// Mitsubishi GX Works2 project: ProjectAtAll1 (1) (2)   PLC: FX3G

// global labels: Global1
VAR_GLOBAL
  Temperature_sensor AT X002 : BOOL;
  Flicking_light3 AT Y003 : BOOL;
  Working_light AT Y007 : BOOL;
  Empty_templets AT X003 : BOOL;
  Melting_Start AT X001 : BOOL;
  Melting_light AT Y001 : BOOL;
  Melting AT Y003 : BOOL;
END_VAR
VAR_GLOBAL CONSTANT
  Nuts_for_Nuts_Mix : REAL := 100;
  Pistachio_for_Nuts_Mix : REAL := 100;
  Nuts_for_Dubai_Chocolate : REAL := 20;
  Pistachio_for_Dubai_Chocolate : REAL := 120;
  Kadaif_for_Dubai_Chocolate : REAL := 60;
END_VAR
VAR_GLOBAL
  Choose_choclate_type AT X004 : BOOL;
END_VAR
VAR_GLOBAL CONSTANT
  Min_Input : INT;
END_VAR
VAR_GLOBAL
  Is_Nuts_Mix AT M150 : BOOL;
  Save_Analog AT D1180 : REAL;
  Analog_Input_1 AT D8280 : INT;
  Analog_Output_2 : BOOL;
  Nuts_Stock AT D1800 : REAL;
  Pistachio_Stock AT D1810 : REAL;
  Kadaif_Stock AT D1820 : REAL;
END_VAR
VAR_GLOBAL CONSTANT
  Melting_Container : REAL := 400;
END_VAR
VAR_GLOBAL
  New_Melting_Container AT D1200 : REAL;
  Empty_templete_sensor AT M3 : BOOL;
END_VAR
VAR_GLOBAL CONSTANT
  Trayes : INT := 4;
END_VAR
VAR_GLOBAL
  Mold_light AT Y002 : BOOL;
END_VAR
VAR_GLOBAL CONSTANT
  Times : INT := 40;
END_VAR
VAR_GLOBAL
  Pass_to_cold_system AT X006 : BOOL;
  Melting_Amount AT D1220 : REAL;
  Not_Enough_Stock AT M7 : BOOL;
  Start_day AT X007 : BOOL;
  Emergency_button AT X005 : BOOL;
  End_the_day AT M5 : BOOL;
  Initial_chocolate AT D1300 : REAL;
  Initial_nuts AT D1310 : REAL;
  Initial_pistachio AT D1320 : REAL;
  Initial_kadaif AT D1330 : REAL;
  Chocolate_Stock AT D1830 : REAL;
END_VAR
VAR_GLOBAL CONSTANT
  Min_Chocolat_Coins : REAL := 400;
END_VAR
VAR_GLOBAL
  Melting_Indicator AT M380 : BOOL;
  Mold_time AT TS4 : BOOL;
  Molding_four_seconds AT TC4 : BOOL;
END_VAR
VAR_GLOBAL CONSTANT
  Div_400_choclate_grams : REAL := 400;
END_VAR
VAR_GLOBAL
  Chocolate_Picked AT D1840 : REAL;
END_VAR
VAR_GLOBAL CONSTANT
  Dubai_Condition_At_Least_6 : REAL := 6;
  Nuts_Mix_Condition_Max_Val : REAL;
END_VAR
VAR_GLOBAL
  Dubai_Picked AT M6 : BOOL;
  Nuts_Mix_Picked AT M5 : BOOL;
END_VAR
VAR_GLOBAL CONSTANT
  Dubai_Condition_At_Least_5 : REAL := 5;
END_VAR
VAR_GLOBAL
  Dubai_chocolate_filling AT D1900 : REAL;
  Nuts_mix_chacolate_filling AT D1910 : REAL;
  Is_Working AT Y007 : BOOL;
  Filling_timer4 AT TC2 : BOOL;
  Filling_timer3 AT TC1 : BOOL;
END_VAR
VAR_GLOBAL CONSTANT
  Five_Second : INT := 50;
END_VAR
VAR_GLOBAL
  Filling_time AT TC1 : BOOL;
  Filling_time1 AT TS1 : BOOL;
  Filling_time2 AT TS2 : BOOL;
  Flicking_light4 AT Y004 : BOOL;
  Flickering_light_index AT M0 : BOOL;
  Count_five_seconds AT TC6 : BOOL;
END_VAR
VAR_GLOBAL CONSTANT
  half_of_Second : INT := 5;
END_VAR
VAR_GLOBAL
  Finish_five_seconds AT TS6 : BOOL;
  Dubai_choclate_frizzing AT D1500 : REAL;
  Nuts_mix_chocolate_frizzing AT D1510 : REAL;
  Freezing_three_seconds AT TC7 : BOOL;
END_VAR
VAR_GLOBAL CONSTANT
  Three_seconds_waiting : INT := 30;
END_VAR
VAR_GLOBAL
  Freezing_time AT TS7 : BOOL;
  Freezing_light AT Y006 : BOOL;
  Packeging_mechine AT D1600 : REAL;
  Dubai_packeging_mechine AT D1600 : REAL;
  Nuts_packeging_mechine AT D1610 : REAL;
END_VAR
VAR_GLOBAL CONSTANT
  Equals_four : REAL := 4;
END_VAR
VAR_GLOBAL
  Dubai_chocolata_bar AT D1700 : REAL;
  Nuts_chocolata_bar AT D1710 : REAL;
  Switch_choclate_table AT X000 : BOOL;
  End_package_light AT Y005 : BOOL;
  Dubai_package AT D1400 : REAL;
  Nuts_mix_package AT D1410 : REAL;
  Package_counter AT CC1 : BOOL;
END_VAR
VAR_GLOBAL CONSTANT
  Four_bars_for_package : INT := 4;
END_VAR
VAR_GLOBAL
  Package_indicator AT M10 : BOOL;
END_VAR
VAR_GLOBAL CONSTANT
  Zero : INT;
END_VAR
VAR_GLOBAL
  Package_indicator2 AT M11 : BOOL;
  Finish_freezing_indicator AT M8 : BOOL;
END_VAR
VAR_GLOBAL CONSTANT
  Three_bars_for_package : INT := 3;
END_VAR
VAR_GLOBAL
  Bars_in_package AT CN1 : INT;
  Package_ready AT CC1 : BOOL;
  Number_of_packages AT D1940 : REAL;
END_VAR
VAR_GLOBAL CONSTANT
  One_package : REAL := 1;
END_VAR
VAR_GLOBAL
  Finish_one_package AT M12 : BOOL;
  End_of_the_day_index AT M13 : BOOL;
END_VAR
VAR_GLOBAL CONSTANT
  Multipy_by_fourty : REAL := 40;
END_VAR
VAR_GLOBAL
  Number_of_packages_output AT D1950 : REAL;
  Analog_Output AT D8282 : INT;
END_VAR

// task Task_01 (event TRUE, interval 0, priority 31): POU_01

PROGRAM POU_01
VAR
  Analog_Output_1 : BOOL;
END_VAR
VAR CONSTANT
  Five_Seconds : INT := 50;
  half_Second : INT := 5;
END_VAR
(* structured ladder/FBD written out as ST: instructions are called as NAME(EN, inputs, outputs); _pN, _eN, _tN stand for wires *)
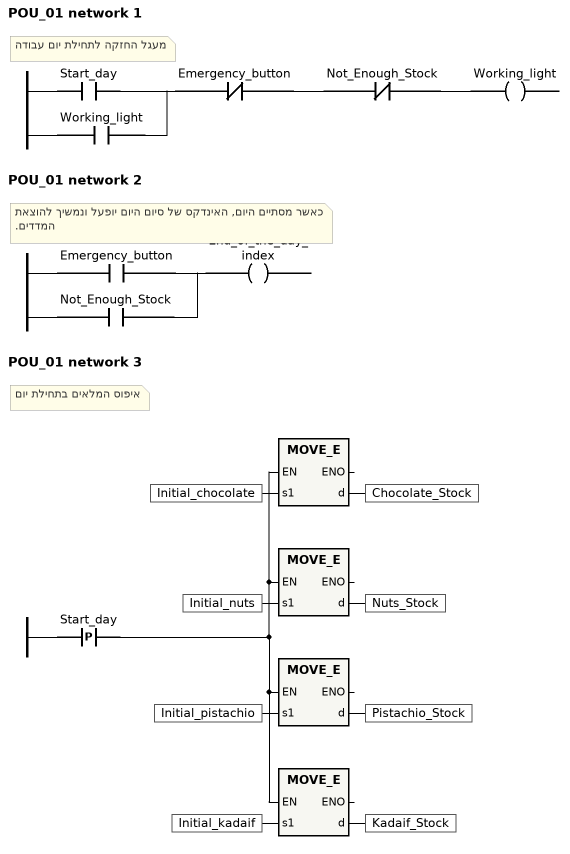
(* network 1 *)
(* מעגל החזקה לתחילת יום עבודה *)
Working_light := ((Start_day OR Working_light) AND NOT Emergency_button) AND NOT Not_Enough_Stock;
(* network 2 *)
(* כאשר מסתיים היום, האינדקס של סיום היום יופעל ונמשיך להוצאת המדדים. *)
End_of_the_day_index := Emergency_button OR Not_Enough_Stock;
(* network 3 *)
(* איפוס המלאים בתחילת יום *)
_p1 := LDP(TRUE, Start_day);
MOVE_E(_p1, Initial_chocolate, Chocolate_Stock);
MOVE_E(_p1, Initial_nuts, Nuts_Stock);
MOVE_E(_p1, Initial_pistachio, Pistachio_Stock);
MOVE_E(_p1, Initial_kadaif, Kadaif_Stock);
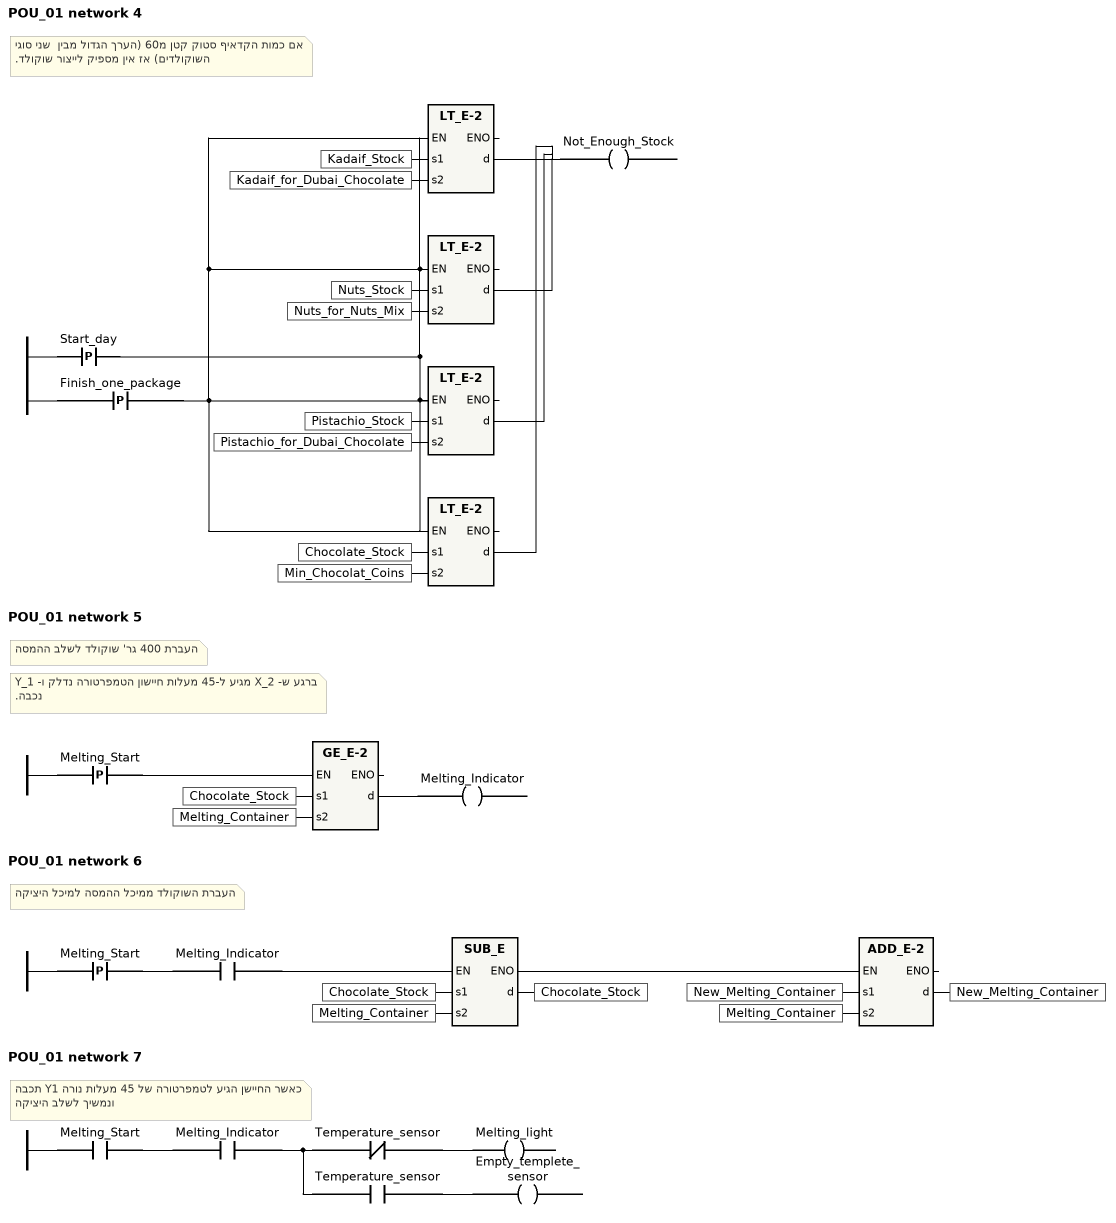
(* network 4 *)
(* אם כמות הקדאיף סטוק קטן מ60 (הערך הגדול מבין  שני סוגי השוקולדים) אז אין מספיק לייצור שוקולד. *)
_p1 := LDP(TRUE, Start_day) OR LDP(TRUE, Finish_one_package);
LT_E(_p1, Kadaif_Stock, Kadaif_for_Dubai_Chocolate, _t2);
LT_E(_p1, Nuts_Stock, Nuts_for_Nuts_Mix, _t3);
LT_E(_p1, Pistachio_Stock, Pistachio_for_Dubai_Chocolate, _t4);
LT_E(_p1, Chocolate_Stock, Min_Chocolat_Coins, _t5);
Not_Enough_Stock := _t2 OR _t3 OR _t4 OR _t5;
(* network 5 *)
(* העברת 400 גר' שוקולד לשלב ההמסה *)
(* ברגע ש- X_2 מגיע ל-45 מעלות חיישון הטמפרטורה נדלק ו- Y_1 נכבה. *)
GE_E(LDP(TRUE, Melting_Start), Chocolate_Stock, Melting_Container, _t1);
Melting_Indicator := _t1;
(* network 6 *)
(* העברת השוקולד ממיכל ההמסה למיכל היציקה *)
_e1 := SUB_E(LDP(TRUE, Melting_Start) AND Melting_Indicator, Chocolate_Stock, Melting_Container, Chocolate_Stock);
ADD_E(_e1, New_Melting_Container, Melting_Container, New_Melting_Container);
(* network 7 *)
(* כאשר החיישן הגיע לטמפרטורה של 45 מעלות נורה Y1 תכבה ונמשיך לשלב היציקה *)
_p1 := Melting_Start AND Melting_Indicator;
Melting_light := _p1 AND NOT Temperature_sensor;
Empty_templete_sensor := _p1 AND Temperature_sensor;
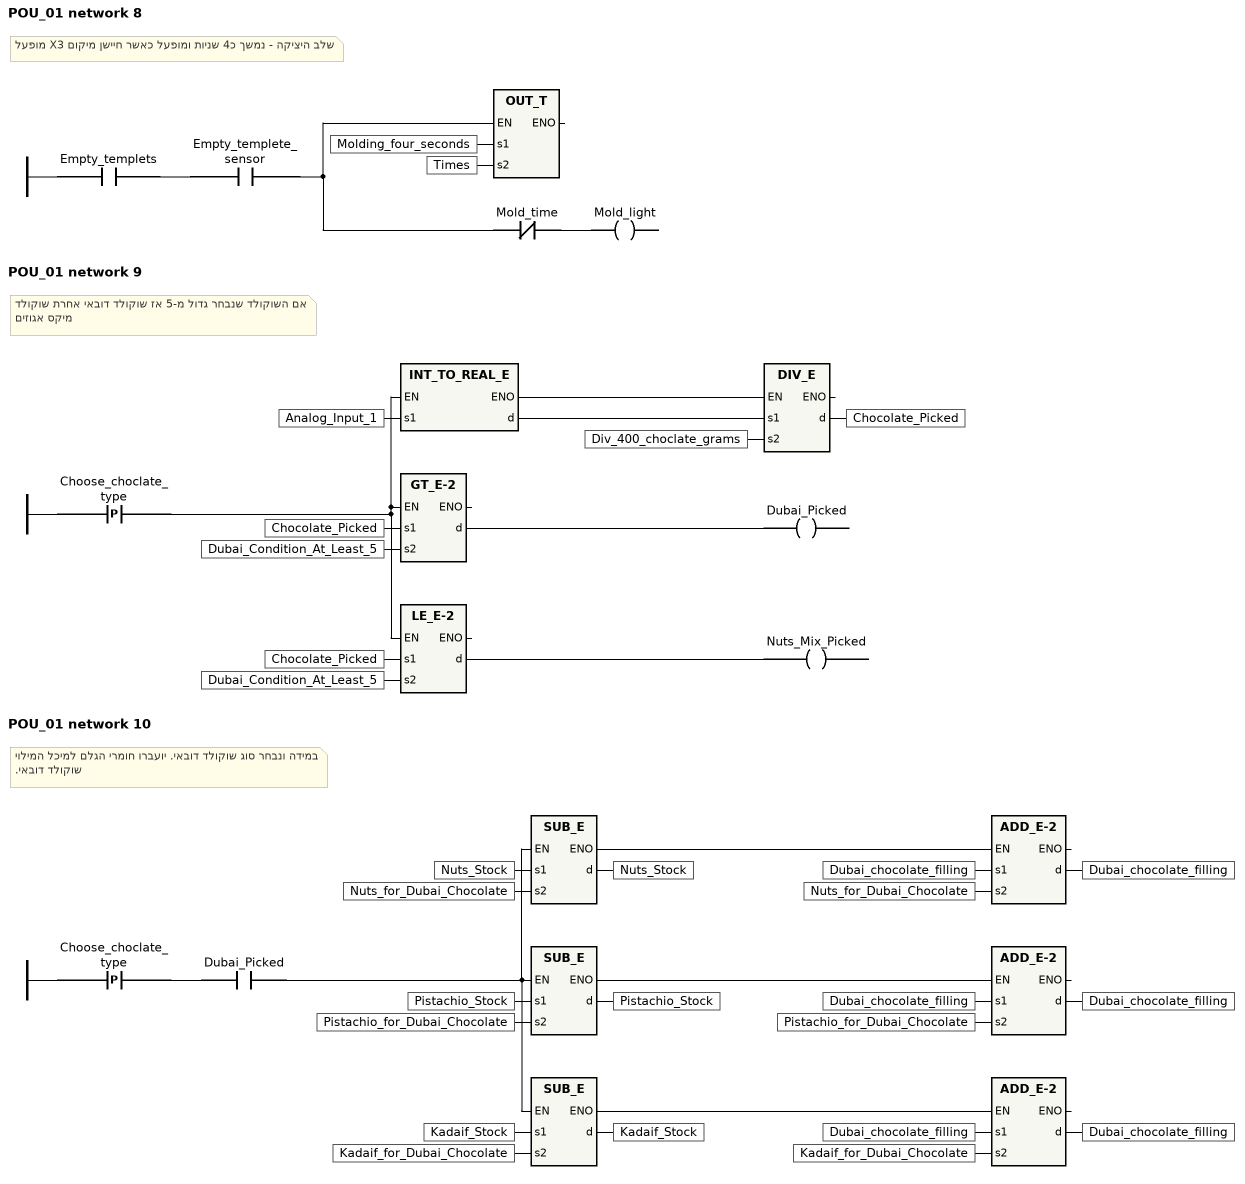
(* network 8 *)
(* שלב היציקה - נמשך כ4 שניות ומופעל כאשר חיישן מיקום X3 מופעל *)
_p1 := Empty_templets AND Empty_templete_sensor;
OUT_T(_p1, Molding_four_seconds, Times);
Mold_light := _p1 AND NOT Mold_time;
(* network 9 *)
(* אם השוקולד שנבחר גדול מ-5 אז שוקולד דובאי אחרת שוקולד מיקס אגוזים *)
_p1 := LDP(TRUE, Choose_choclate_type);
_e3 := INT_TO_REAL_E(_p1, Analog_Input_1, _t2);
DIV_E(_e3, _t2, Div_400_choclate_grams, Chocolate_Picked);
GT_E(_p1, Chocolate_Picked, Dubai_Condition_At_Least_5, _t4);
Dubai_Picked := _t4;
LE_E(_p1, Chocolate_Picked, Dubai_Condition_At_Least_5, _t5);
Nuts_Mix_Picked := _t5;
(* network 10 *)
(* במידה ונבחר סוג שוקולד דובאי. יועברו חומרי הגלם למיכל המילוי שוקולד דובאי. *)
_p1 := LDP(TRUE, Choose_choclate_type) AND Dubai_Picked;
_e2 := SUB_E(_p1, Nuts_Stock, Nuts_for_Dubai_Chocolate, Nuts_Stock);
ADD_E(_e2, Dubai_chocolate_filling, Nuts_for_Dubai_Chocolate, Dubai_chocolate_filling);
_e3 := SUB_E(_p1, Pistachio_Stock, Pistachio_for_Dubai_Chocolate, Pistachio_Stock);
ADD_E(_e3, Dubai_chocolate_filling, Pistachio_for_Dubai_Chocolate, Dubai_chocolate_filling);
_e4 := SUB_E(_p1, Kadaif_Stock, Kadaif_for_Dubai_Chocolate, Kadaif_Stock);
ADD_E(_e4, Dubai_chocolate_filling, Kadaif_for_Dubai_Chocolate, Dubai_chocolate_filling);
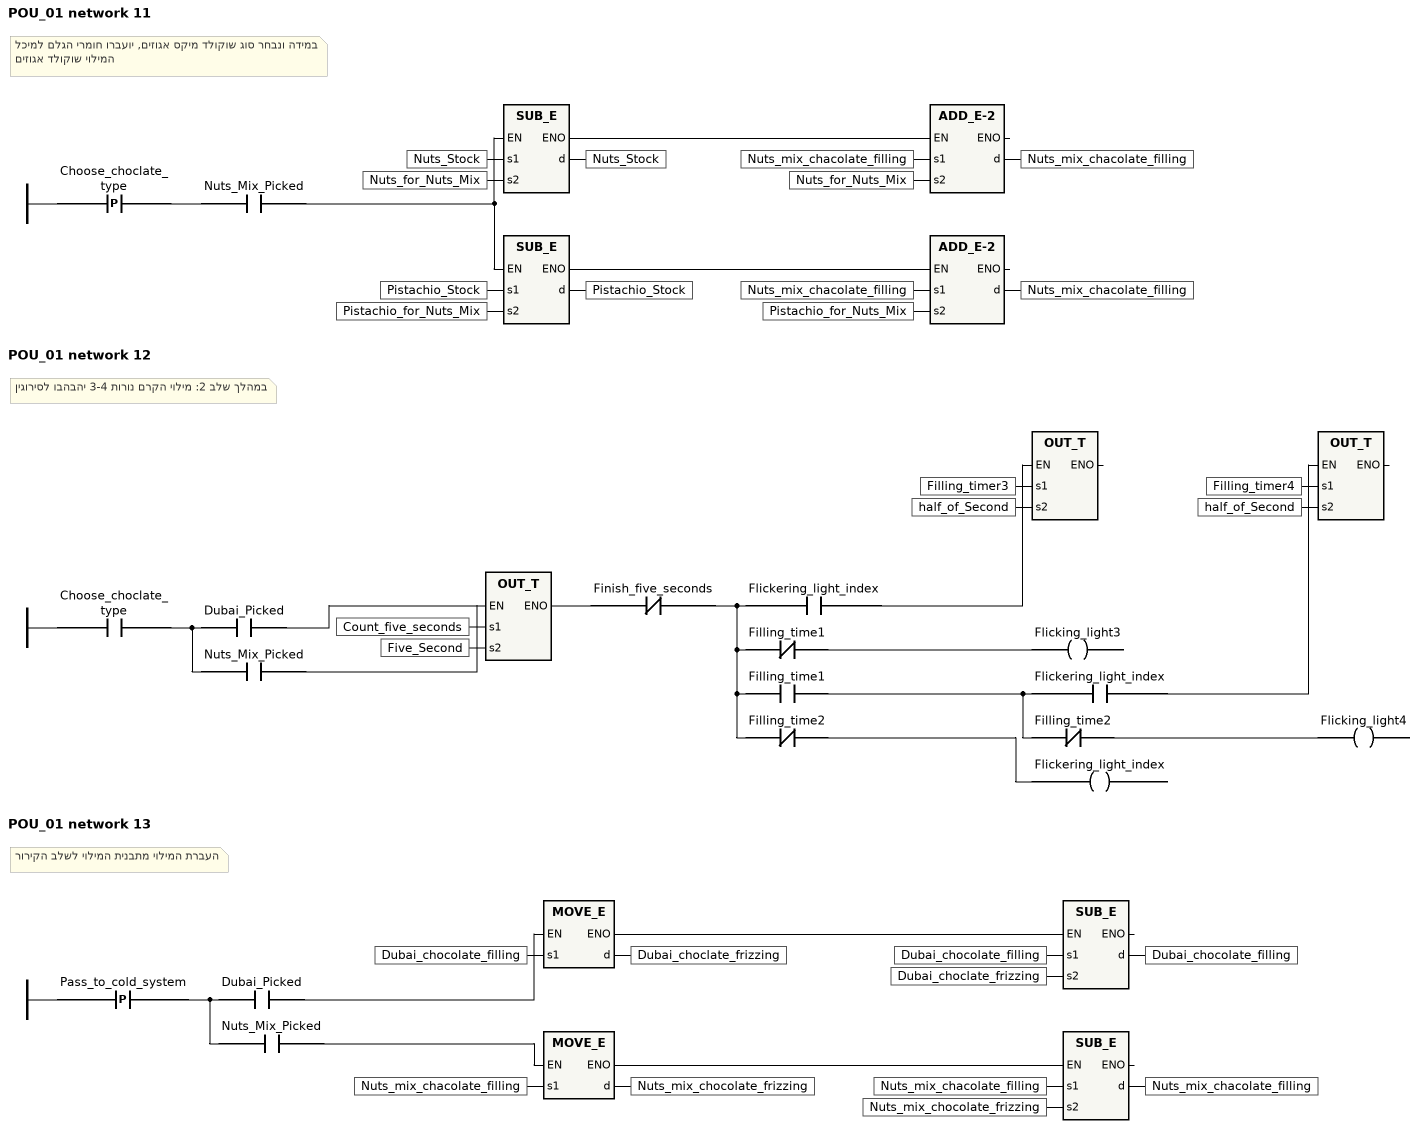
(* network 11 *)
(* במידה ונבחר סוג שוקולד מיקס אגוזים, יועברו חומרי הגלם למיכל המילוי שוקולד אגוזים *)
_p1 := LDP(TRUE, Choose_choclate_type) AND Nuts_Mix_Picked;
_e2 := SUB_E(_p1, Nuts_Stock, Nuts_for_Nuts_Mix, Nuts_Stock);
ADD_E(_e2, Nuts_mix_chacolate_filling, Nuts_for_Nuts_Mix, Nuts_mix_chacolate_filling);
_e3 := SUB_E(_p1, Pistachio_Stock, Pistachio_for_Nuts_Mix, Pistachio_Stock);
ADD_E(_e3, Nuts_mix_chacolate_filling, Pistachio_for_Nuts_Mix, Nuts_mix_chacolate_filling);
(* network 12 *)
(* במהלך שלב 2: מילוי הקרם נורות 3-4 יהבהבו לסירוגין *)
_e1 := OUT_T((Choose_choclate_type AND Dubai_Picked) OR (Choose_choclate_type AND Nuts_Mix_Picked), Count_five_seconds, Five_Second);
_p2 := _e1 AND NOT Finish_five_seconds;
OUT_T(_p2 AND Flickering_light_index, Filling_timer3, half_of_Second);
Flicking_light3 := _p2 AND NOT Filling_time1;
_p3 := _p2 AND Filling_time1;
OUT_T(_p3 AND Flickering_light_index, Filling_timer4, half_of_Second);
Flicking_light4 := _p3 AND NOT Filling_time2;
Flickering_light_index := _p2 AND NOT Filling_time2;
(* network 13 *)
(* העברת המילוי מתבנית המילוי לשלב הקירור *)
_p1 := LDP(TRUE, Pass_to_cold_system);
_e2 := MOVE_E(_p1 AND Dubai_Picked, Dubai_chocolate_filling, Dubai_choclate_frizzing);
SUB_E(_e2, Dubai_chocolate_filling, Dubai_choclate_frizzing, Dubai_chocolate_filling);
_e3 := MOVE_E(_p1 AND Nuts_Mix_Picked, Nuts_mix_chacolate_filling, Nuts_mix_chocolate_frizzing);
SUB_E(_e3, Nuts_mix_chacolate_filling, Nuts_mix_chocolate_frizzing, Nuts_mix_chacolate_filling);
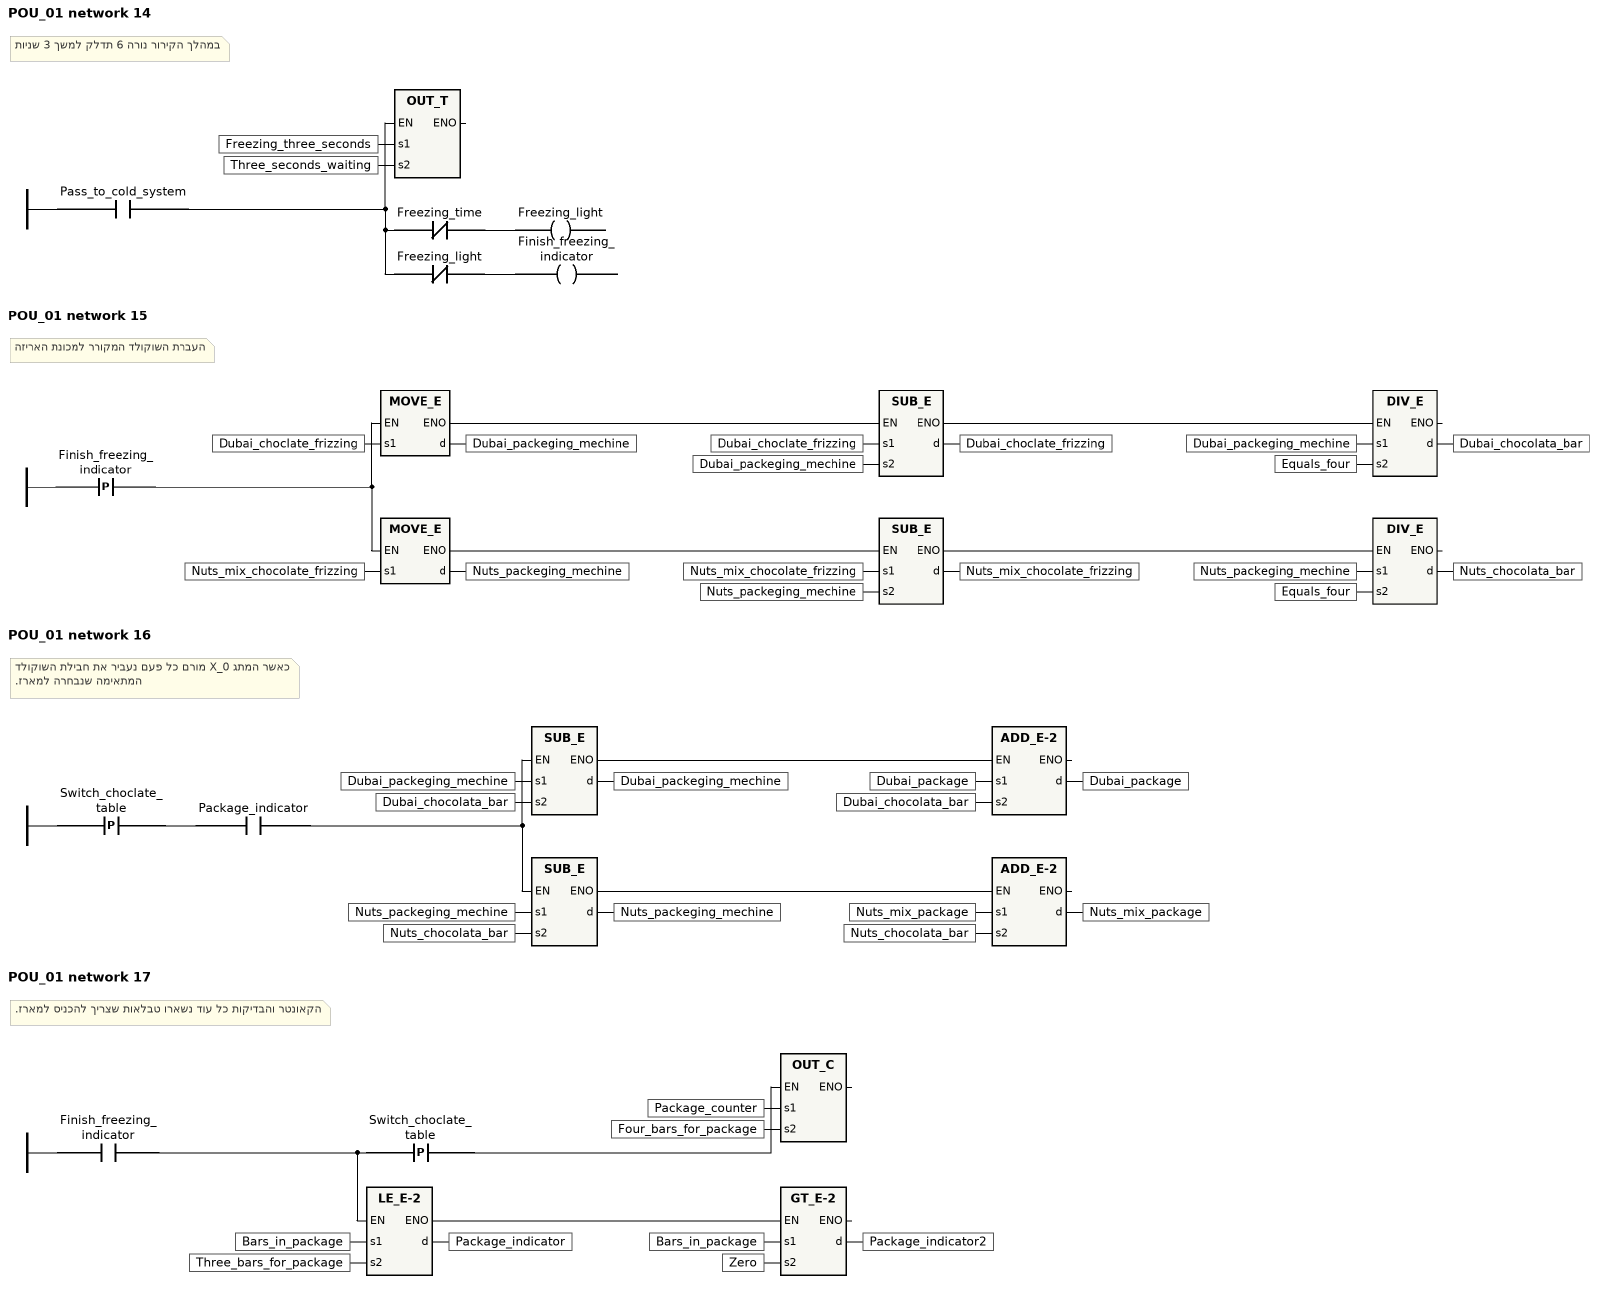
(* network 14 *)
(* במהלך הקירור נורה 6 תדלק למשך 3 שניות *)
OUT_T(Pass_to_cold_system, Freezing_three_seconds, Three_seconds_waiting);
Freezing_light := Pass_to_cold_system AND NOT Freezing_time;
Finish_freezing_indicator := Pass_to_cold_system AND NOT Freezing_light;
(* network 15 *)
(* העברת השוקולד המקורר למכונת האריזה *)
_p1 := LDP(TRUE, Finish_freezing_indicator);
_e2 := MOVE_E(_p1, Dubai_choclate_frizzing, Dubai_packeging_mechine);
_e3 := SUB_E(_e2, Dubai_choclate_frizzing, Dubai_packeging_mechine, Dubai_choclate_frizzing);
DIV_E(_e3, Dubai_packeging_mechine, Equals_four, Dubai_chocolata_bar);
_e4 := MOVE_E(_p1, Nuts_mix_chocolate_frizzing, Nuts_packeging_mechine);
_e5 := SUB_E(_e4, Nuts_mix_chocolate_frizzing, Nuts_packeging_mechine, Nuts_mix_chocolate_frizzing);
DIV_E(_e5, Nuts_packeging_mechine, Equals_four, Nuts_chocolata_bar);
(* network 16 *)
(* כאשר המתג X_0 מורם כל פעם נעביר את חבילת השוקולד המתאימה שנבחרה למארז. *)
_p1 := LDP(TRUE, Switch_choclate_table) AND Package_indicator;
_e2 := SUB_E(_p1, Dubai_packeging_mechine, Dubai_chocolata_bar, Dubai_packeging_mechine);
ADD_E(_e2, Dubai_package, Dubai_chocolata_bar, Dubai_package);
_e3 := SUB_E(_p1, Nuts_packeging_mechine, Nuts_chocolata_bar, Nuts_packeging_mechine);
ADD_E(_e3, Nuts_mix_package, Nuts_chocolata_bar, Nuts_mix_package);
(* network 17 *)
(* הקאונטר והבדיקות כל עוד נשארו טבלאות שצריך להכניס למארז. *)
OUT_C(Finish_freezing_indicator AND LDP(TRUE, Switch_choclate_table), Package_counter, Four_bars_for_package);
_e1 := LE_E(Finish_freezing_indicator, Bars_in_package, Three_bars_for_package, Package_indicator);
GT_E(_e1, Bars_in_package, Zero, Package_indicator2);
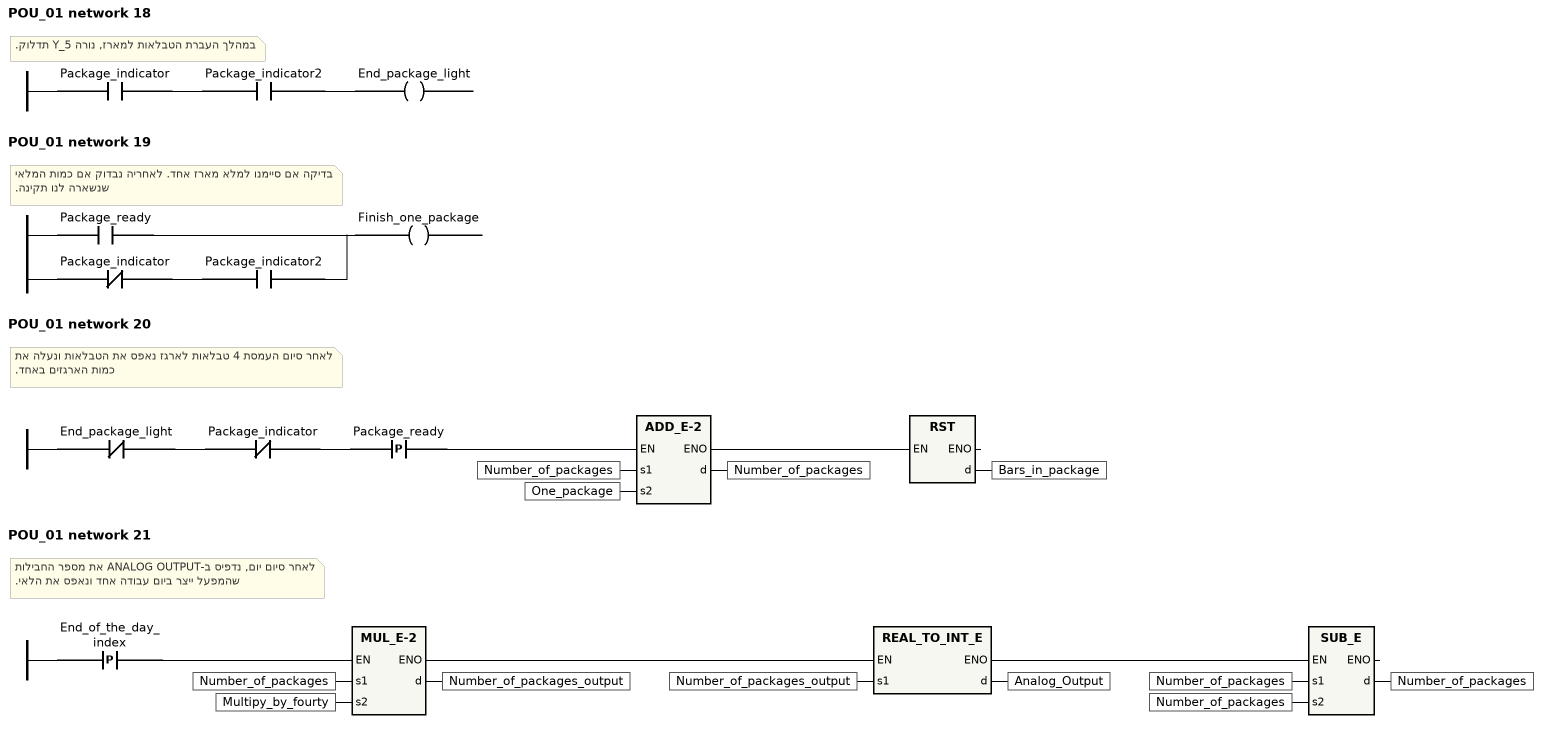
(* network 18 *)
(* במהלך העברת הטבלאות למארז, נורה Y_5 תדלוק. *)
End_package_light := Package_indicator AND Package_indicator2;
(* network 19 *)
(* בדיקה אם סיימנו למלא מארז אחד. לאחריה נבדוק אם כמות המלאי שנשארה לנו תקינה. *)
Finish_one_package := Package_ready OR (NOT Package_indicator AND Package_indicator2);
(* network 20 *)
(* לאחר סיום העמסת 4 טבלאות לארגז נאפס את הטבלאות ונעלה את כמות הארגזים באחד. *)
_e1 := ADD_E(NOT End_package_light AND NOT Package_indicator AND LDP(TRUE, Package_ready), Number_of_packages, One_package, Number_of_packages);
RST(_e1, Bars_in_package);
(* network 21 *)
(* לאחר סיום יום, נדפיס ב-ANALOG OUTPUT את מספר החבילות שהמפעל ייצר ביום עבודה אחד ונאפס את הלאי. *)
_e1 := MUL_E(LDP(TRUE, End_of_the_day_index), Number_of_packages, Multipy_by_fourty, Number_of_packages_output);
_e2 := REAL_TO_INT_E(_e1, Number_of_packages_output, Analog_Output);
SUB_E(_e2, Number_of_packages, Number_of_packages, Number_of_packages);
END_PROGRAM
